PROGRAM MAIN
VAR
	fbDriveNc 	: FB_DriveNC;
	fbDriveCan	: FB_DriveCAN;
	iDrive		: I_DriveBase := fbDriveNc;
	
	// Drive Swap Control
	bNcDrive: BOOL;
	bCANDrive: BOOL;
END_VAR

IF bNcDrive THEN
	bNcDrive := FALSE;
	iDrive := fbDriveNc;
END_IF

IF bCANDrive THEN
	bCANDrive := FALSE;
	iDrive := fbDriveCan;
END_IF


iDrive.Enable();

END_PROGRAM

(* stored: Version 1.1.0.1, ProductVersion 3.1.4024.6
   POU MAIN: Id {0ddc26d6-86f9-4c1c-a4d5-6fbbe034d1d7}, SpecialFunc None *)
